RoboDK station: Projekt.rdk

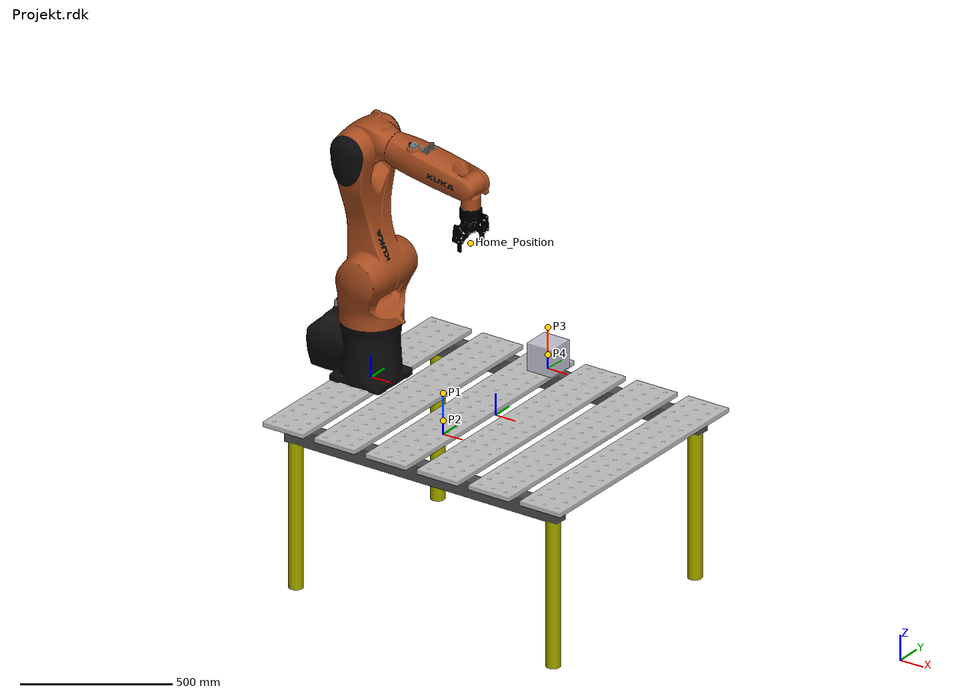
[picture v0: the station drawn from its stored meshes, robots at their saved joint values, targets as dots, program paths as lines]
Station Projekt (saved by RoboDK 5.2.1). Poses are relative to the parent item; angles as X-Y-Z fixed-axis rotations.
  - frame KUKA KR 10 R900 sixx Base at (-500, 0, 0) mm
    - robot KUKA KR 10 R900 sixx: 6 axes, payload 10 kg, reach 901 mm, repeatability 0.03 mm, weight 52 kg
        modified DH rows (alpha deg, a mm, theta deg, d mm): 0, 0, 0, 400; -90, 25, 0, 0; 0, 455, -90, 0; -90, 35, 0, 420; 90, 0, 0, 0; -90, 0, 180, 80
        joint limits [-170, -190, -120, -185, -120, -350] to [170, 45, 156, 185, 120, 350]; home [0, -90, 90, 0, 0, 0]; saved at [0, -95.584, 106.182, 0, 79.402, -280]
      - tool Gripper RobotiQ 85 Opened, TCP at (0, 0, 130) mm, size 147.4 x 146.8 x 75 mm
  - frame Baza at (0, 0, 0) mm
    - object Table at (0, 0, 0) mm, size 1193.8 x 965.2 x 609.6 mm, geometry from welding_table.sld
    - target Home_Position (Cartesian target) at (-100, 0, 600) mm, rotated rx 180 ry 0 rz -100 deg; joints [0, -95.584, 106.182, 0, 79.402, -280] of KUKA KR 10 R900 sixx
  - frame Part_1 at (0, -300, 50) mm
    - target P1 (Cartesian target) at (0, 0, 150) mm, rotated rx 180 ry 0 rz -180 deg; joints [30.964, -48.861, 105.748, 0, 33.113, -329.036] of KUKA KR 10 R900 sixx
    - target P2 (Cartesian target) at (0, 0, 50) mm, rotated rx 180 ry 0 rz 180 deg; joints [30.964, -38.123, 104.533, 0, 23.59, -329.036] of KUKA KR 10 R900 sixx
  - frame Part_2 at (0, 300, 50) mm
    - target P3 (Cartesian target) at (0, 0, 150) mm, rotated rx -180 ry 0 rz 180 deg; joints [-30.964, -48.861, 105.748, -180, -33.113, -210.964] of KUKA KR 10 R900 sixx
    - target P4 (Cartesian target) at (0, 0, 50) mm, rotated rx -180 ry 0 rz -180 deg; joints [-30.964, -38.123, 104.533, -180, -23.59, -210.964] of KUKA KR 10 R900 sixx
    - object box at (0, 0, 50) mm, size 100 x 100 x 100 mm, geometry from box.sld
  - program Restore (1 instructions, listed below)
  - program Pick_Part_1 (6 instructions, listed below)
  - program Place_Part_2 (6 instructions, listed below)
  - program MainProgram (8 instructions, listed below)
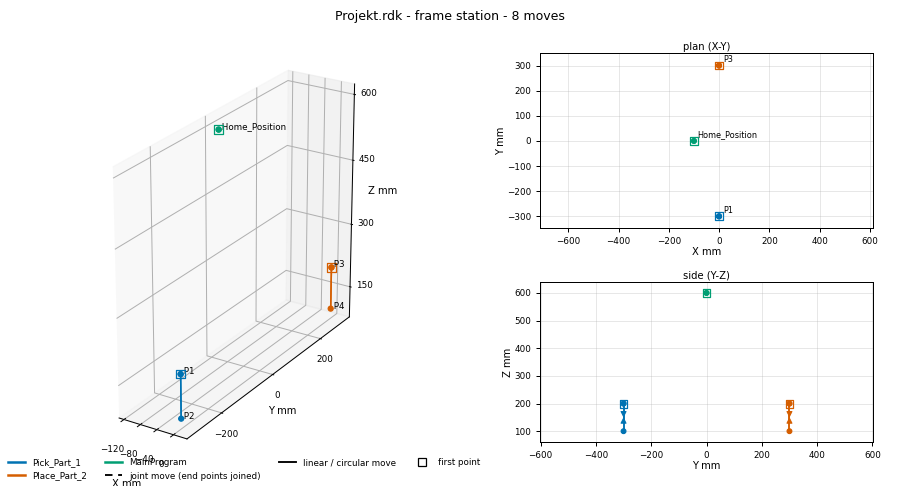
[picture p0: tool path of Projekt.rdk in frame station, 8 of 8 moves have a stored position in this frame; points joined in program order, loops and branches not executed]

--- program Restore (robot KUKA KR 10 R900 sixx) ---
  Replace objects

--- program Pick_Part_1 (robot KUKA KR 10 R900 sixx) ---
  Set Ref.: Part_1
  Set Tool: Gripper RobotiQ 85 Opened
  MoveJ (P1)
  MoveL (P2)
  Attach to Gripper RobotiQ 85 Opened
  MoveL (P1)

--- program Place_Part_2 (robot KUKA KR 10 R900 sixx) ---
  Set Ref.: Part_2
  Set Tool: Gripper RobotiQ 85 Opened
  MoveJ (P3)
  MoveL (P4)
  Detach from Gripper RobotiQ 85 Opened
  MoveL (P3)

--- program MainProgram (robot KUKA KR 10 R900 sixx) ---
  Set Ref.: Base_Mesa -> Baza
  Set Tool: Gripper RobotiQ 85 Opened
  MoveJ (Home_Position)
  Call Pick_Part_1
  Call Place_Part_2
  Set Ref.: Base_Mesa -> Baza
  MoveJ (Home_Position)
  Call Program1
